SYSTEM TANK_MVCL (* Level Control System Model+View+Control+HMI *)
  (* Standard: 61499-1; Classification: Simulation; ApplicationDomain: Process Control *)
  (* Version 0.1, 2004-09-013, JHC, Rockwell Automation, Extended from TANK_MVL. *)
  (* Version 0.0, 2004-09-03, JHC, Rockwell Automation, Extended from TANK_MVL. *)
  APPLICATION TANK_CTL (* Tank Control Application *)
    FBS
      FACE : FACEPLATE;
      CTRL : FB_PIDR;
      RECORDER : STRIP4;
      CLK : E_CYCLE;
      T_MDL : TANK_MDL;
      PUMP_SPEED : FB_SLIDER;
      OUT_UINT : FB_REAL_UINT;
      PV_UINT : FB_REAL_UINT;
    END_FBS
    EVENT_CONNECTIONS
      CLK.EO TO CTRL.REQ;
      CTRL.CNF TO OUT_UINT.REQ;
      T_MDL.EO TO PV_UINT.REQ;
      OUT_UINT.CNF TO RECORDER.REQ;
      CTRL.CNF TO FACE.REQ;
    END_CONNECTIONS
    DATA_CONNECTIONS
      FACE.SP TO CTRL.SP;
      FACE.SP TO CTRL.X0;
      PUMP_SPEED.OUT TO T_MDL.DRAW;
      CTRL.XOUT TO T_MDL.FEED;
      T_MDL.LEVEL TO CTRL.PV;
      T_MDL.LEVEL TO FACE.PV;
      CTRL.XOUT TO FACE.XOUT;
      PUMP_SPEED.OUT TO RECORDER.PEN1;
      FACE.SP TO RECORDER.PEN2;
      CTRL.XOUT TO OUT_UINT.IN;
      OUT_UINT.OUT TO RECORDER.PEN3;
      T_MDL.LEVEL TO PV_UINT.IN;
      PV_UINT.OUT TO RECORDER.PEN4;
    END_CONNECTIONS
  END_APPLICATION
  DEVICE HMI : FRAME_DEVICE
    RESOURCE RECORDER : PANEL_RESOURCE
      FBS
        PUMP_SPEED : SUBL_1;
        PV : SUBL_1;
        OUT : SUBL_1;
        RECORDER : STRIP4;
        PV_UINT : FB_REAL_UINT;
        OUT_UINT : FB_REAL_UINT;
        SP : SUBL_1;
      END_FBS
      EVENT_CONNECTIONS
        PV.IND TO PV_UINT.REQ;
        OUT.IND TO OUT_UINT.REQ;
        START.COLD TO PV.INIT;
        START.WARM TO PV.INIT;
        RECORDER.INITO TO SP.INIT;
        PV.INITO TO PUMP_SPEED.INIT;
        PUMP_SPEED.INITO TO OUT.INIT;
        OUT.INITO TO RECORDER.INIT;
        OUT_UINT.CNF TO RECORDER.REQ;
      END_CONNECTIONS
      DATA_CONNECTIONS
        SP.RD_1 TO RECORDER.PEN2;
        [red,orange,green,blue] TO RECORDER.COLORS;
        COLOR#lightGray TO RECORDER.BKGD;
        [200,150] TO RECORDER.SIZE;
        1 TO RECORDER.DX;
        PUMP_SPEED.RD_1 TO RECORDER.PEN1;
        PV.RD_1 TO PV_UINT.IN;
        OUT.RD_1 TO OUT_UINT.IN;
        OUT_UINT.OUT TO RECORDER.PEN3;
        PV_UINT.OUT TO RECORDER.PEN4;
      END_CONNECTIONS
    END_RESOURCE
    RESOURCE PUMP : PANEL_RESOURCE
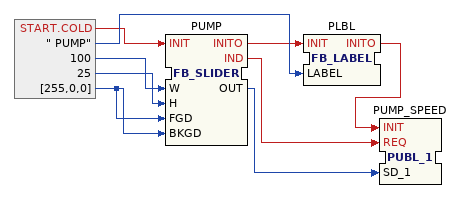
      FBS
        PUMP_SPEED : PUBL_1;
        PUMP : FB_SLIDER;
        PLBL : FB_LABEL;
      END_FBS
      EVENT_CONNECTIONS
        PUMP.INITO TO PLBL.INIT;
        PLBL.INITO TO PUMP_SPEED.INIT;
        START.COLD TO PUMP.INIT;
        PUMP.IND TO PUMP_SPEED.REQ;
      END_CONNECTIONS
      DATA_CONNECTIONS
        " PUMP" TO PLBL.LABEL;
        100 TO PUMP.W;
        25 TO PUMP.H;
        PUMP.OUT TO PUMP_SPEED.SD_1;
        [255,0,0] TO PUMP.FGD;
        [255,0,0] TO PUMP.BKGD;
      END_CONNECTIONS
    END_RESOURCE
  END_DEVICE
  DEVICE CONTROLLER : FRAME_DEVICE
    RESOURCE FACE : PANEL_RESOURCE
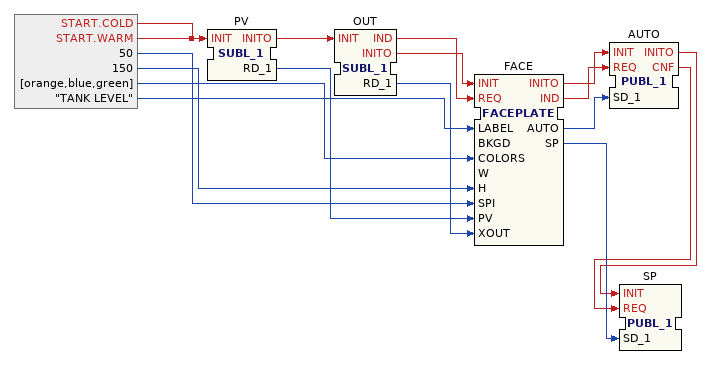
      FBS
        PV : SUBL_1;
        FACE : FACEPLATE;
        SP : PUBL_1;
        OUT : SUBL_1;
        AUTO : PUBL_1;
      END_FBS
      EVENT_CONNECTIONS
        START.COLD TO PV.INIT;
        START.WARM TO PV.INIT;
        OUT.IND TO FACE.REQ;
        FACE.INITO TO AUTO.INIT;
        FACE.IND TO AUTO.REQ;
        AUTO.INITO TO SP.INIT;
        AUTO.CNF TO SP.REQ;
        PV.INITO TO OUT.INIT;
        OUT.INITO TO FACE.INIT;
      END_CONNECTIONS
      DATA_CONNECTIONS
        PV.RD_1 TO FACE.PV;
        50 TO FACE.SPI;
        150 TO FACE.H;
        FACE.SP TO SP.SD_1;
        OUT.RD_1 TO FACE.XOUT;
        FACE.AUTO TO AUTO.SD_1;
        [orange,blue,green] TO FACE.COLORS;
        "TANK LEVEL" TO FACE.LABEL;
      END_CONNECTIONS
    END_RESOURCE
    RESOURCE CTL : EMB_RES
      FBS
        CLK : E_CYCLE;
        PV : SUBL_1;
        SP : SUBL_1;
        CTRL : FB_PIDR;
        OUT : PUBL_1;
        AUTO : SUBL_1;
      END_FBS
      EVENT_CONNECTIONS
        START.COLD TO SP.INIT;
        START.WARM TO SP.INIT;
        SP.INITO TO PV.INIT;
        PV.INITO TO AUTO.INIT;
        AUTO.INITO TO OUT.INIT;
        CTRL.CNF TO OUT.REQ;
        CLK.EO TO CTRL.REQ;
        START.STOP TO CLK.STOP;
        OUT.INITO TO CLK.START;
      END_CONNECTIONS
      DATA_CONNECTIONS
        t#250 ms TO CLK.DT;
        5 TO CTRL.KP;
        CTRL.XOUT TO OUT.SD_1;
        SP.RD_1 TO CTRL.SP;
        PV.RD_1 TO CTRL.PV;
        AUTO.RD_1 TO CTRL.AUTO;
        SP.RD_1 TO CTRL.X0;
        t#250ms TO CTRL.DT;
        t#2s TO CTRL.TR;
        t#0s TO CTRL.TD;
      END_CONNECTIONS
    END_RESOURCE
  END_DEVICE
  DEVICE MV : FRAME_DEVICE (* Model+View *)
    RESOURCE TANK_MDL : EMB_RES
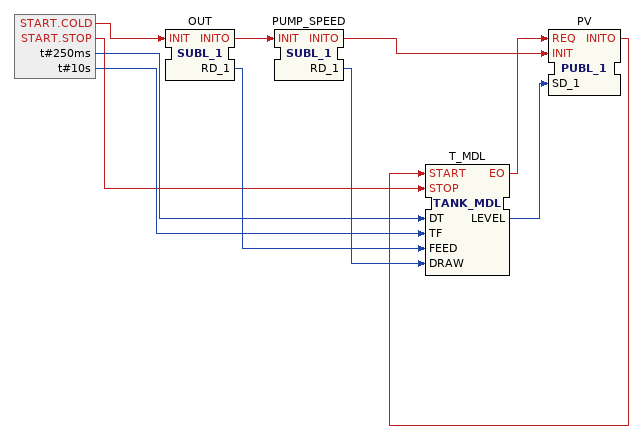
      FBS
        T_MDL : TANK_MDL;
        PUMP_SPEED : SUBL_1;
        OUT : SUBL_1;
        PV : PUBL_1;
      END_FBS
      EVENT_CONNECTIONS
        START.COLD TO OUT.INIT;
        OUT.INITO TO PUMP_SPEED.INIT;
        T_MDL.EO TO PV.REQ;
        START.STOP TO T_MDL.STOP;
        PUMP_SPEED.INITO TO PV.INIT;
        PV.INITO TO T_MDL.START;
      END_CONNECTIONS
      DATA_CONNECTIONS
        PUMP_SPEED.RD_1 TO T_MDL.DRAW;
        t#250ms TO T_MDL.DT;
        OUT.RD_1 TO T_MDL.FEED;
        t#10s TO T_MDL.TF;
        T_MDL.LEVEL TO PV.SD_1;
      END_CONNECTIONS
    END_RESOURCE
    RESOURCE PUMP_MDL : EMB_RES
      FBS
        P_MDL : SHAFT_MDL;
        PUMP_POS : PUBL_1;
        PUMP_SPEED : SUBL_1;
        UNSC : UNSCALE;
      END_FBS
      EVENT_CONNECTIONS
        START.COLD TO PUMP_SPEED.INIT;
        PUMP_SPEED.INITO TO PUMP_POS.INIT;
        P_MDL.EO TO PUMP_POS.REQ;
        PUMP_POS.INITO TO P_MDL.START;
        PUMP_SPEED.IND TO UNSC.REQ;
      END_CONNECTIONS
      DATA_CONNECTIONS
        t#100ms TO P_MDL.DT;
        P_MDL.POS TO PUMP_POS.SD_1;
        UNSC.OUT TO P_MDL.V;
        PUMP_SPEED.RD_1 TO UNSC.IN;
        360 TO UNSC.MAX;
      END_CONNECTIONS
    END_RESOURCE
    RESOURCE VALVE : VIEW_PANEL
      FBS
        OUT : SUBL_1;
        VALVE : VALVE_VIEW;
        OUT_UINT : FB_REAL_UINT;
      END_FBS
      EVENT_CONNECTIONS
        START.COLD TO OUT.INIT;
        OUT.INITO TO VALVE.INIT;
        OUT.IND TO OUT_UINT.REQ;
        OUT_UINT.CNF TO VALVE.REQ;
      END_CONNECTIONS
      DATA_CONNECTIONS
        50 TO VALVE.DIA;
        [0,255,0] TO VALVE.FGD;
        OUT.RD_1 TO OUT_UINT.IN;
        OUT_UINT.OUT TO VALVE.POS;
      END_CONNECTIONS
    END_RESOURCE
    RESOURCE TANK : VIEW_PANEL
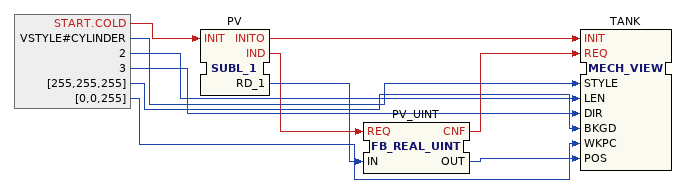
      FBS
        TANK : MECH_VIEW;
        PV : SUBL_1;
        PV_UINT : FB_REAL_UINT;
      END_FBS
      EVENT_CONNECTIONS
        PV.INITO TO TANK.INIT;
        START.COLD TO PV.INIT;
        PV.IND TO PV_UINT.REQ;
        PV_UINT.CNF TO TANK.REQ;
      END_CONNECTIONS
      DATA_CONNECTIONS
        VSTYLE#CYLINDER TO TANK.STYLE;
        2 TO TANK.LEN;
        3 TO TANK.DIR;
        [255,255,255] TO TANK.BKGD;
        [0,0,255] TO TANK.WKPC;
        PV.RD_1 TO PV_UINT.IN;
        PV_UINT.OUT TO TANK.POS;
      END_CONNECTIONS
    END_RESOURCE
    RESOURCE PUMP : VIEW_PANEL
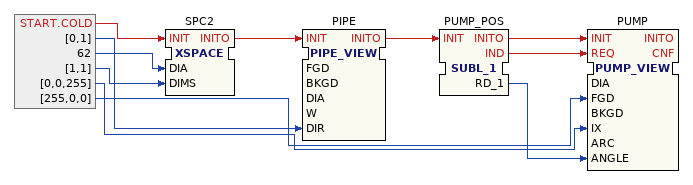
      FBS
        PUMP_POS : SUBL_1;
        SPC2 : XSPACE;
        PIPE : PIPE_VIEW;
        PUMP : PUMP_VIEW;
      END_FBS
      EVENT_CONNECTIONS
        SPC2.INITO TO PIPE.INIT;
        START.COLD TO SPC2.INIT;
        PIPE.INITO TO PUMP_POS.INIT;
        PUMP_POS.INITO TO PUMP.INIT;
        PUMP_POS.IND TO PUMP.REQ;
      END_CONNECTIONS
      DATA_CONNECTIONS
        [0,1] TO PIPE.DIR;
        62 TO SPC2.DIA;
        [1,1] TO SPC2.DIMS;
        PUMP_POS.RD_1 TO PUMP.ANGLE;
        [0,0,255] TO PUMP.IX;
        [255,0,0] TO PUMP.FGD;
      END_CONNECTIONS
    END_RESOURCE
    DATA_CONNECTIONS
      [1,2] TO TANK.SIZE;
      75 TO TANK.DIA;
      50 TO PUMP.DIA;
      [4,1] TO PUMP.SIZE;
      50 TO VALVE.DIA;
      [1,3] TO VALVE.SIZE;
    END_CONNECTIONS
  END_DEVICE
  DATA_CONNECTIONS (* parameter values *)
    [240,100,210,270] TO HMI.BOUNDS;
    [450,100,175,270] TO MV.BOUNDS;
    [100,100,140,270] TO CONTROLLER.BOUNDS;
  END_CONNECTIONS
END_SYSTEM
